{attribute 'qualified_only'}
VAR_GLOBAL
	//data to THIS station/machine to be accepted
	ToStation: typeRemote;
	
	//data fed to NEXT or supervisor segment station
	//todo

END_VAR

(* stored: Version 1.1.0.1, ProductVersion 3.1.4024.12
   GVL Remote: Id {0cd9502d-d5ea-4a11-87aa-63e44e107acf} *)
